PROGRAM LoadFromAGV
VAR
	// Default
	Done: BOOL;
	
	// Container
	InvalidAGVPart: BOOL;
	ContainerColor: STRING;
	Debug: BOOL;
END_VAR

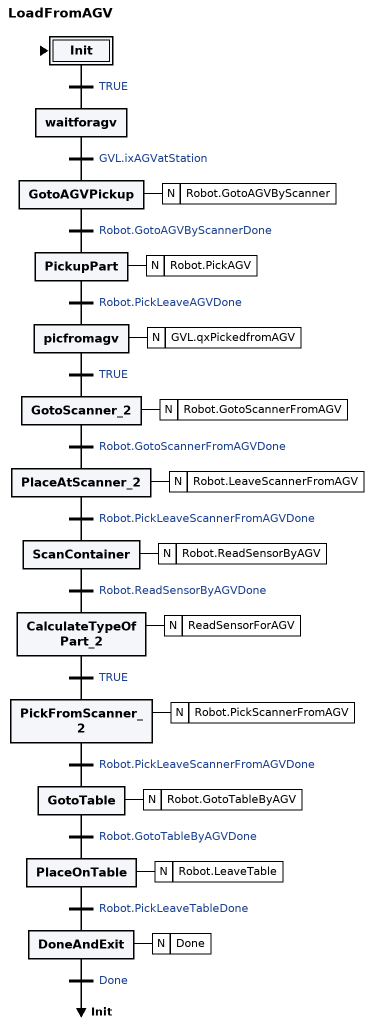
INITIAL_STEP Init:
END_STEP
TRANSITION FROM Init TO waitforagv
    := TRUE;
END_TRANSITION
STEP waitforagv:
END_STEP
TRANSITION FROM waitforagv TO GotoAGVPickup
    := GVL.ixAGVatStation;
END_TRANSITION
STEP GotoAGVPickup:
    Robot.GotoAGVByScanner(N);
END_STEP
TRANSITION FROM GotoAGVPickup TO PickupPart
    := Robot.GotoAGVByScannerDone;
END_TRANSITION
STEP PickupPart:
    Robot.PickAGV(N);
END_STEP
TRANSITION FROM PickupPart TO picfromagv
    := Robot.PickLeaveAGVDone;
END_TRANSITION
STEP picfromagv:
    GVL.qxPickedfromAGV(N);
END_STEP
TRANSITION FROM picfromagv TO GotoScanner_2
    := TRUE;
END_TRANSITION
STEP GotoScanner_2:
    Robot.GotoScannerFromAGV(N);
END_STEP
TRANSITION FROM GotoScanner_2 TO PlaceAtScanner_2
    := Robot.GotoScannerFromAGVDone;
END_TRANSITION
STEP PlaceAtScanner_2:
    Robot.LeaveScannerFromAGV(N);
END_STEP
TRANSITION FROM PlaceAtScanner_2 TO ScanContainer
    := Robot.PickLeaveScannerFromAGVDone;
END_TRANSITION
STEP ScanContainer:
    Robot.ReadSensorByAGV(N);
END_STEP
TRANSITION FROM ScanContainer TO CalculateTypeOfPart_2
    := Robot.ReadSensorByAGVDone;
END_TRANSITION
STEP CalculateTypeOfPart_2:
    ReadSensorForAGV(N);
END_STEP
TRANSITION FROM CalculateTypeOfPart_2 TO PickFromScanner_2
    := TRUE;
END_TRANSITION
STEP PickFromScanner_2:
    Robot.PickScannerFromAGV(N);
END_STEP
TRANSITION FROM PickFromScanner_2 TO GotoTable
    := Robot.PickLeaveScannerFromAGVDone;
END_TRANSITION
STEP GotoTable:
    Robot.GotoTableByAGV(N);
END_STEP
TRANSITION FROM GotoTable TO PlaceOnTable
    := Robot.GotoTableByAGVDone;
END_TRANSITION
STEP PlaceOnTable:
    Robot.LeaveTable(N);
END_STEP
TRANSITION FROM PlaceOnTable TO DoneAndExit
    := Robot.PickLeaveTableDone;
END_TRANSITION
STEP DoneAndExit:
    Done(N);
END_STEP
TRANSITION FROM DoneAndExit TO Init
    := Done;
END_TRANSITION

ACTION ReadSensorForAGV:
ContainerColor := Robot.IdentifyPartFB.Color;
IF Robot.IdentifyPartFB.Product <> 'CONTAINER' THEN
	GVL.mwStationStatus := 1000;
	GVL.ixEmergencyStop := TRUE;
END_IF
END_ACTION

ACTION SkipScan:
ContainerColor:= 'RED';
Debug:= TRUE;
END_ACTION

END_PROGRAM

(* stored: Version 1.1.0.1, ProductVersion 3.1.4024.12
   POU LoadFromAGV: Id {06c3c9a7-52d0-4ea6-8d09-a992c42cb347}, SpecialFunc None
   Action ReadSensorForAGV: Id {f37e4d7d-a527-4e54-b8de-5ae89553c237}
   Action SkipScan: Id {b7141d62-f827-4e7b-936b-55e1f2d2d4a7} *)
